// TIA Portal project "Conveyor_Sorting_System" (V17)

(* hardware
DEVICE "S7-1500/ET200MP station_1"  S7-1500 station
   slot 0: "Rail_0"  Rack  6ES7 590-1***0-0AA0
   slot 1: "PLC_1"  CPU 1511-1 PN  6ES7 511-1AK02-0AB0  V2.9
      slot 3: "CPU display_1"  6ES7591-1AA00-0AA0
      slot 32768: "PROFINET interface_1"  X1
         slot 32769: "Port_1"  X1 P1
         slot 32770: "Port_2"  X1 P2
      slot 34817: "Virtual CP interface port_1"  Virtual CP interface port  Virtual CP interface port
DEVICE "ET 200SP station_1"  ET 200SP-Station
   slot 0: "Rack_0"  Rack  6ES5 710-8MAx1
   slot 0: "IO device_1"  IM 155-6 PN ST  6ES7 155-6AU01-0BN0  V4.2
   slot 1: "Server module_1"  Server module  6ES7 193-6PA00-0AA0  V1.1
      slot 1: "Server module_1"  Server module
   slot 127: "BA 2xRJ45"  BA 2xRJ45  6ES7 193-6AR00-0AA0  V0.0
      slot 1: "Port_1"  X1 P1 R  6ES7 193-6AR00-0AA0  V0.0
      slot 2: "Port_2"  X1 P2 R  6ES7 193-6AR00-0AA0  V0.0
DEVICE "HMI_1"  KTP700 Basic PN
   slot 0: "HMI_1"  KTP700 Basic PN  6AV2 123-2GB03-0AX0  17.0.0.0
   slot 1: "HMI_RT_1"  KTP700 Basic PN  6AV2 123-2GB03-0AX0  17.0.0.0
   slot 5: "HMI_1.IE_CP_1"  PROFINET Interface  17.0.0.0
      slot 1: "PROFINET Interface_1"  PROFINET Interface
         slot 1: "Port_1"  Port
*)

// ===== PLC "PLC_1"  CPU 1511-1 PN =====

TYPE "Package_UDT"
   STRUCT
      PackageID : Int;
      Weight : Real;
      Destination : Int;
      Timestamp : Date_And_Time;
      IsValid : Bool;
      FaultCode : Int;
   END_STRUCT;
END_TYPE

DATA_BLOCK "ProductBuffer_DB"   // DB1
{ S7_Optimized_Access := 'TRUE' }
VERSION : 0.1
   VAR
      PackageBuffer : Array[0..9] of "Package_UDT";
   END_VAR
BEGIN
END_DATA_BLOCK

DATA_BLOCK "FB_ConveyorZone_DB"   // DB2
{ S7_Optimized_Access := 'TRUE' }
VERSION : 0.1
// stored: InstanceOfName FB_ConveyorZone
"FB_ConveyorZone"
BEGIN
END_DATA_BLOCK

FUNCTION_BLOCK "FB_ConveyorZone"   // FB1, SCL
{ S7_Optimized_Access := 'TRUE' }
VERSION : 0.1
   VAR_INPUT
      xEnable : Bool;
      xEmergencyStop : Bool;
      xSensorEntry : Bool;
      xSensorExit : Bool;
      rPackageWeight : Real;
   END_VAR
   VAR_OUTPUT
      xMotorRun : Bool;
      xFault : Bool;
      xZoneReady : Bool;
      iCurrentState : Int;
      sFaultMessage : String;
   END_VAR
   VAR
      iState : Int;
      xLastSensor : Bool;
   END_VAR
BEGIN
   // State Machine
   // 0=IDLE, 1=RUNNING, 2=STOPPING, 3=FAULT, 4=EMERGENCY
   CASE #iState OF

       0: // IDLE
           #xMotorRun := FALSE;
           #xZoneReady := TRUE;
           #xFault := FALSE;
           #sFaultMessage := 'IDLE - Waiting';
           IF #xEnable AND NOT #xEmergencyStop THEN
               #iState := 1;
           END_IF;
           IF #xEmergencyStop THEN
               #iState := 4;
           END_IF;

       1: // RUNNING
           #xMotorRun := TRUE;
           #xZoneReady := FALSE;
           #sFaultMessage := 'RUNNING - Package in transit';
           IF #xEmergencyStop THEN
               #iState := 4;
           END_IF;
           IF #rPackageWeight > 50.0 THEN
               #sFaultMessage := 'FAULT - Weight limit exceeded';
               #iState := 3;
           END_IF;
           IF #xSensorExit THEN
               #iState := 2;
           END_IF;

       2: // STOPPING
           #xMotorRun := FALSE;
           #sFaultMessage := 'STOPPING - Package delivered';
           IF NOT #xSensorExit THEN
               #iState := 0;
           END_IF;

       3: // FAULT
           #xMotorRun := FALSE;
           #xFault := TRUE;
           #xZoneReady := FALSE;
           #sFaultMessage := 'FAULT - Operator reset required';
           IF #xEnable AND NOT #xEmergencyStop THEN
               #iState := 0;
           END_IF;

       4: // EMERGENCY STOP
           #xMotorRun := FALSE;
           #xFault := TRUE;
           #xZoneReady := FALSE;
           #sFaultMessage := 'E-STOP ACTUATED - Safety interlock active';

   END_CASE;

   #iCurrentState := #iState;
END_FUNCTION_BLOCK

ORGANIZATION_BLOCK "Main"   // OB1, LAD, ProgramCycle
TITLE = "Main Program Sweep (Cycle)"
{ S7_Optimized_Access := 'TRUE' }
VERSION : 0.1
   VAR_INPUT
      Initial_Call : Bool;   // Initial call of this OB
      Remanence : Bool;   // =True, if remanent data are available
   END_VAR
BEGIN

REGION Network 1: FB_ConveyorZone_DB
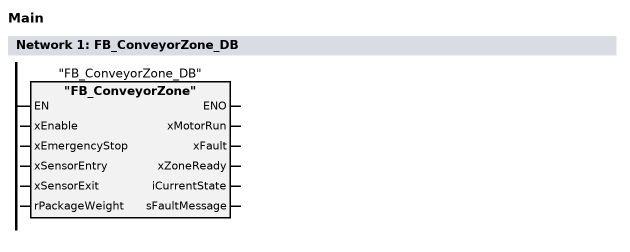
   RUNG wire#powerrail
      "FB_ConveyorZone_DB"(xEnable :=, xEmergencyStop :=, xSensorEntry :=, xSensorExit :=, rPackageWeight :=, xMotorRun =>, xFault =>, xZoneReady =>, iCurrentState =>, sFaultMessage =>)
   END_RUNG
   // the same network as SCL:
   "FB_ConveyorZone_DB"();   // "FB_ConveyorZone"
END_REGION
END_ORGANIZATION_BLOCK

(* ===== HMI "HMI_RT_1" =====
system functions are stored by id; their names below are inferred from use
connection "HMI_Connection_1": ETHERNET, SMART_S7_1500_OMS

HMI tags "Default tag table"
   "Tag_ScreenNumber" : UInt, internal

HMI tags "Conveyor_Tags"
   "Zone1_State" : Int = PLC FB_ConveyorZone_DB.iCurrentState AT %DB1.DBW0, 1 s
   "Zone1_Fault" : Bool = PLC FB_ConveyorZone_DB.xFault AT %DB1.DBW0, 1 s
   "Zone1_Motor" : Bool = PLC FB_ConveyorZone_DB.xMotorRun AT %DB1.DBX0.0, 1 s
   "Zone1_FaultMsg" : String[254] = PLC FB_ConveyorZone_DB.sFaultMessage AT %DB1.DBX0.0, 1 s
   "Zone1_Enable" : Bool = PLC FB_ConveyorZone_DB.xEnable AT %DB1.DBX0.0, 1 s
   "Zone1_EStop" : Bool = PLC FB_ConveyorZone_DB.xEmergencyStop AT %DB1.DBX0.0, 1 s
   "PackageWeight" : Real = PLC FB_ConveyorZone_DB.rPackageWeight AT %DB1.DBX0.0, 1 s

Template "Template_1" 800x480
   Button "Exit" at 714,429 size 71x50; TextOff 'Exit'; PictureOff "ExitRuntime_KTP700_Basic_PN_TR"; PictureOn "ExitRuntime_KTP700_Basic_PN_TR"
      on Release: StopRuntime(0)
   Button "Template_Button" at 614,429 size 71x50; TextOff 'Text'
   Button "Template_Button_1" at 514,429 size 71x50; TextOff 'Text'
   Button "Template_Button_2" at 414,429 size 71x50; TextOff 'Text'
   Button "Template_Button_3" at 314,429 size 71x50; TextOff 'Text'
   Button "Template_Button_4" at 214,429 size 71x50; TextOff 'Text'
   Button "Template_Button_5" at 114,429 size 71x50; TextOff 'Text'
   Button "Start screen" at 14,429 size 71x50; TextOff 'Start screen'; PictureOff "NavigateHome_KTP700_Basic_PN_TR"; PictureOn "NavigateHome_KTP700_Basic_PN_TR"
      on Release: ActivateScreen("Root screen", 0)
   SymbolicIOField "Symbolic_IO_Field_Screen" at 93,9 size 600x33; TextOff '0'; TextOn '1'; TextList "TextList_ScreenNames"
      ProcessValue <- "Tag_ScreenNumber"
      on Change: ActivateScreenByNumber("Tag_ScreenNumber", 0)
   DateTimeField "HmiScreenItemData" at 695,25 size 105x25
   DateTimeField "HmiScreenItemData_1" at 695,0 size 105x25
   GraphicView "Logo" at 0,0 size 91x51; Picture "Logo of HMI_1"

screen "Root screen" 800x480, template "Template_1"
   on GenerateScreen: SetTag("Tag_ScreenNumber", 1)
   TextField "HmiScreenItemData" at 82,85 size 654x53; Text 'Welcome to Raj Bag HMI_1 (KTP700 Basic+ PN)!'
   Circle "Circle_1" at 100,214 size 34x34
      Appearance <- "Zone1_State"
   IOField "I/O field_1" at 260,217 size 96x32; FormatPattern ????????????????????????????????????????????????????????????????????????????????
      ProcessValue <- "Zone1_FaultMsg"
   IOField "I/O field_2" at 454,217 size 96x32; FormatPattern 999.9
      ProcessValue <- "PackageWeight"
   Button "Button_1" at 642,217 size 96x32; TextOff 'E-STOP'
      on Click: SetBit("Zone1_EStop")
   Button "Button_2" at 317,310 size 139x32; TextOff 'START ZONE'
      on Click: SetBit("Zone1_Enable")
   TextField "Text field_1" at 157,274 size 69x23; Text 'Text'
   TextField "Text field_2" at 69,257 size 123x23; Text 'ZONE 1 STATE'
   TextField "Text field_3" at 237,257 size 141x23; Text 'FAULT MESSAGE'
   TextField "Text field_4" at 403,256 size 196x23; Text 'PACKAGE WEIGHT (kg)'
   TextField "Text field_5" at 642,255 size 94x23; Text 'CONTROLS'
*)